{attribute addProperty BoxType "EL6201-0000-0017"}
{attribute addProperty Id "Slave_16A_DO0BIT10.125121Slave_16A_DO1BIT10.125122Slave_16A_DO2BIT10.125123Slave_16A_DO3BIT10.125124Slave_16B_DO0BIT10.125125Slave_16B_DO1BIT10.125126Slave_16B_DO2BIT10.125127Slave_16B_DO3BIT10.125128"}
{attribute addProperty CRC "1903651203"}
{attribute addProperty SizeInBites "8"}
{attribute addProperty SizeInBytes "1"}
TYPE Slave_16_Outputs_71776983 :
STRUCT
	{attribute addProperty Name "Slave_16A_DO0"}
	Slave_16A_DO0 : BIT;
	{attribute addProperty Name "Slave_16A_DO1"}
	Slave_16A_DO1 : BIT;
	{attribute addProperty Name "Slave_16A_DO2"}
	Slave_16A_DO2 : BIT;
	{attribute addProperty Name "Slave_16A_DO3"}
	Slave_16A_DO3 : BIT;
	{attribute addProperty Name "Slave_16B_DO0"}
	Slave_16B_DO0 : BIT;
	{attribute addProperty Name "Slave_16B_DO1"}
	Slave_16B_DO1 : BIT;
	{attribute addProperty Name "Slave_16B_DO2"}
	Slave_16B_DO2 : BIT;
	{attribute addProperty Name "Slave_16B_DO3"}
	Slave_16B_DO3 : BIT;
END_STRUCT
END_TYPE

(* stored: Version 1.2.0.0, ProductVersion 3.1.4024.9
   DUT Slave_16_Outputs_71776983: Id {a2524228-c378-46ec-93f8-efb78ba7b06f} *)
